PROGRAM C_Machine_CTRL
VAR
	
	bFirstRun					:BOOL;
	bFirstAutoCycle				:BOOL;
	bSmacDone					:BOOL;
	bKistlerDone				:BOOL;
	rSmacDone					:R_TRIG;
	rKistlerDone				:R_TRIG;
	bStatisticsFlag				:ARRAY[0..1] OF BOOL;
	
	eMachineState				:E_MachineState:=E_MachineState.SYSTEM_POWER_UP;

	//Timers && Triggers
	tonSys_Init					:Tc2_Standard.TON:=(PT:=T#1S);
	tonSys_InitTimeout			:Tc2_Standard.TON:=(PT:=T#3M);					
	tonWAIT_SMAC_KISLR			:Tc2_Standard.TON;
	tonFirstAutoCycle			:Tc2_Standard.TON:=(PT:=T#500MS);
	
	//Process Cycle
	eCycleState					:E_ProcessCycle;
	stTotalReport				:ST_ProcessReport;
	bStartConditions			:BOOL;	
	tonTwoHandsTouching			:Tc2_Standard.TON;         
	bScrewPresent				: BOOL;
	bReservoirPresent			: BOOL;
	tonGrippersOpennedSignal	: TON;
	tonDelayExe					:Tc2_Standard.TON:=(PT:=T#100MS);
	rtrigResetModule			:Tc2_Standard.R_TRIG;
	rtrigProcessLogShift		:Tc2_Standard.R_TRIG;
	
	
	//Index
	idx							:INT;
	
END_VAR
//----------------------------------------------------------------------------oldschoo1

// Call for Actions

   b_Machine_Status();		//State machina 
	 c_ProcessCycle();	   //Master sequencer


//----------------------------------------------------------------*


// Process Report circular buffer
rtrigProcessLogShift(CLK:=eCycleState=E_ProcessCycle.Saving_DATA);

IF rtrigProcessLogShift.Q THEN 
	FOR idx:= 250 TO 2 BY -1 DO
		GVL_PERSISTENT.stProccessReportLog[idx]:=GVL_PERSISTENT.stProccessReportLog[idx-1];
	END_FOR
	GVL_PERSISTENT.stProccessReportLog[1]:=stTotalReport;
END_IF//																										||
//--------------------------------------------------------------------------------------------------------oldschoo1

ACTION b_Machine_Status:




//Timers && Triggers
tonSys_Init(IN:=stMachineStatus.bInitialising);
tonSys_InitTimeout(IN:=stMachineStatus.bInitialising);
IF stMachineStatus.eMachineState <> E_MachineState.SYSTEM_AUTO_CYCLE THEN
	bFirstAutoCycle							:= FALSE;
END_IF

//Transition IF Cycle Stop Fault OR Imediate Fault
IF NOT stMasterCtrl.bNoMachineImmediateFault THEN		
				stMachineStatus.eMachineState := E_MachineState.IMMEDIATE_FAULT;
	
ELSIF NOT stMasterCtrl.bNoCycleStopFault AND NOT stMachineStatus.bImmediateStopped THEN
				stMachineStatus.eMachineState := E_MachineState.CYCLE_STOP_FAULT;
END_IF

IF NOT GVL_Master.stMasterCTRL.bManualModeRequest THEN
	CMD_Axis.bManualMode	:=FALSE;
	CMD_Smac.bManualMode	:=FALSE;
	CMD_Kistler.bManualMode	:=FALSE;
END_IF
(****************************************************MACHINE_CTRL*******************************************************************)
//STATE MACHINE: ------------------------------------------------------------------------------------------------------------------SM
CASE stMachineStatus.eMachineState OF

E_MachineState.SYSTEM_POWER_UP: 		// ------------------------------------------------------------------------------POWER_UP

				IF tonSystemPowerUP.Q THEN
						stMachineStatus.eMachineState := E_MachineState.IMMEDIATE_STOPPED;//
				END_IF
	
E_MachineState.IMMEDIATE_STOPPED:		// ---------------------------------------------------------------------IMMEDIATE_STOPPED

				IF stMasterCtrl.bNoMachineImmediateFault AND bResetButtonFallingEdge THEN
						stMachineStatus.eMachineState := E_MachineState.SYSTEM_INITIALISING;//
						
				ELSIF NOT stMasterCtrl.bNoCycleStopFault THEN
						stMachineStatus.eMachineState := E_MachineState.CYCLE_STOP_FAULT;//
					
				ELSIF NOT stMasterCtrl.bNoMachineImmediateFault THEN
					stMachineStatus.eMachineState := E_MachineState.IMMEDIATE_FAULT;//	
				END_IF		


E_MachineState.SYSTEM_INITIALISING:		// -------------------------------------------------------------------SYSTEM_INITIALISING		

				IF tonSys_Init.Q THEN
						CMD_Axis.bEnable	:=TRUE;
						CMD_Smac.bEnable	:=TRUE;
						CMD_Kistler.bEnable	:=TRUE;
						
						CMD_Axis.bAbort		:=FALSE;
						CMD_Smac.bAbort		:=FALSE;
						CMD_Kistler.bAbort	:=FALSE;
				END_IF

				//IF Axis_STATUS.bReady AND Kistler_STATUS.bReady  AND Smac_STATUS.bReady THEN 
				 IF Axis_STATUS.bReady AND Kistler_STATUS.bReady AND ( GVL_PERSISTENT.bSMACEnable AND Smac_STATUS.bReady OR NOT GVL_PERSISTENT.bSMACEnable) THEN //**LAA  29092025
										stMachineStatus.eMachineState:= E_MachineState.SYSTEM_READY_TO_START;//
				END_IF

				IF bStopButtonFallingEdge OR 
			 	  (stMasterCtrl.bNoMachineImmediateFault AND 
			 	  (stMasterCtrl.bCycleStopRequest OR tonSys_InitTimeout.Q) AND 
			       stMasterCtrl.bAllActionsStopped)
					THEN
										stMachineStatus.eMachineState := E_MachineState.CYCLE_STOPPED;//
						
				ELSIF stMasterCtrl.bNoMachineImmediateFault AND NOT stMasterCtrl.bNoCycleStopFault 
					THEN		
										stMachineStatus.eMachineState := E_MachineState.CYCLE_STOP_FAULT;//
			
				ELSIF NOT stMasterCtrl.bNoMachineImmediateFault 
					THEN
										stMachineStatus.eMachineState := E_MachineState.IMMEDIATE_FAULT;//
				END_IF
			
					
E_MachineState.SYSTEM_READY_TO_START:	// -------------------------------------------------------------------SYSTEM_READY_TO_START<<<

				IF 	 bStartButtonFallingEdge AND stMasterCtrl.bAllModulesReady THEN
					
										stMachineStatus.eMachineState := E_MachineState.SYSTEM_AUTO_CYCLE;//
				
				ELSIF bStopButtonFallingEdge THEN
					
										stMachineStatus.eMachineState := E_MachineState.STOPPING;//
										
				ELSIF stMasterCtrl.bNoMachineImmediateFault AND NOT stMasterCtrl.bNoCycleStopFault THEN	
	
										stMachineStatus.eMachineState := E_MachineState.CYCLE_STOP_FAULT;//
			
				ELSIF NOT stMasterCtrl.bNoMachineImmediateFault THEN
										stMachineStatus.eMachineState := E_MachineState.IMMEDIATE_FAULT;//
				ELSIF GVL_Master.stMasterCTRL.bManualModeRequest AND stMasterCtrl.bNoMachineImmediateFault AND stMasterCtrl.bNoCycleStopFault THEN
										stMachineStatus.eMachineState := E_MachineState.MANUAL_MODE;//
				END_IF

				

E_MachineState.SYSTEM_AUTO_CYCLE:		// ---------------------------------------------------------------------SYSTEM_AUTO_CYCLE	

				IF bStopButtonFallingEdge THEN					
										stMachineStatus.eMachineState := E_MachineState.STOPPING;//
						
				ELSIF stMasterCtrl.bCycleStopRequest THEN 
					
										stMachineStatus.eMachineState := E_MachineState.STOPPING;//
										
				ELSIF stMasterCtrl.bNoMachineImmediateFault AND NOT stMasterCtrl.bNoCycleStopFault THEN	
	
										stMachineStatus.eMachineState := E_MachineState.CYCLE_STOP_FAULT;//
			
				ELSIF NOT stMasterCtrl.bNoMachineImmediateFault THEN
										stMachineStatus.eMachineState := E_MachineState.IMMEDIATE_FAULT;//
				END_IF	

E_MachineState.SYSTEM_STANDBY:;//



E_MachineState.STOPPING:				// ------------------------------------------------------------------------------STOPPING

				IF stMasterCtrl.bAllActionsStopped THEN
										stMachineStatus.eMachineState := E_MachineState.CYCLE_STOPPED;//					
				END_IF
				CMD_Axis.bEnable	:=FALSE;
				CMD_Smac.bEnable	:=FALSE;
				CMD_Kistler.bEnable	:=FALSE;
				
				CMD_Axis.bAbort		:=TRUE;
				CMD_Smac.bAbort		:=TRUE;
				CMD_Kistler.bAbort	:=TRUE;

E_MachineState.CYCLE_STOPPED:			// -------------------------------------------------------------------------CYCLE_STOPPED

				IF stMasterCtrl.bNoCycleStopFault   AND 
	      		NOT stMasterCtrl.bCycleStopRequest  AND 
                               bResetButtonFallingEdge

									THEN	
										stMachineStatus.eMachineState := E_MachineState.SYSTEM_INITIALISING;		
				END_IF	

E_MachineState.IMMEDIATE_FAULT:			// -----------------------------------------------------------------------IMMEDIATE_FAULT
				
				CMD_Axis.bEnable	:=FALSE;
				CMD_Smac.bEnable	:=FALSE;
				CMD_Kistler.bEnable	:=FALSE;
						
				CMD_Axis.bAbort		:=TRUE;
				CMD_Smac.bAbort		:=TRUE;
				CMD_Kistler.bAbort	:=TRUE;
				
				IF stMasterCtrl.bNoMachineImmediateFault	THEN
										stMachineStatus.eMachineState := E_MachineState.IMMEDIATE_STOPPED;		
				END_IF

E_MachineState.CYCLE_STOP_FAULT:		// ----------------------------------------------------------------------CYCLE_STOP_FAULT

				CMD_Axis.bEnable	:=FALSE;
				CMD_Smac.bEnable	:=FALSE;
				CMD_Kistler.bEnable	:=FALSE;
						
				CMD_Axis.bAbort		:=TRUE;
				CMD_Smac.bAbort		:=TRUE;
				CMD_Kistler.bAbort	:=TRUE;
				
				IF stMasterCtrl.bNoCycleStopFault THEN
										stMachineStatus.eMachineState := E_MachineState.CYCLE_STOPPED;
				END_IF	


E_MachineState.MANUAL_MODE:;//

				IF bStopButtonFallingEdge OR NOT GVL_Master.stMasterCTRL.bManualModeRequest THEN
					
										stMachineStatus.eMachineState := E_MachineState.STOPPING;//
										
										CMD_Axis.bManualMode:=FALSE;
										CMD_Smac.bManualMode:=FALSE;
										CMD_Kistler.bManualMode:=FALSE;
										CMD_Axis.bAbort		:=TRUE;
										CMD_Smac.bAbort		:=TRUE;
										CMD_Kistler.bAbort	:=TRUE;
				ELSIF stMasterCtrl.bNoMachineImmediateFault AND NOT stMasterCtrl.bNoCycleStopFault THEN	
	
										stMachineStatus.eMachineState := E_MachineState.CYCLE_STOP_FAULT;//
										
										CMD_Axis.bManualMode:=FALSE;
										CMD_Smac.bManualMode:=FALSE;
										CMD_Kistler.bManualMode:=FALSE;
										CMD_Axis.bAbort		:=TRUE;
										CMD_Smac.bAbort		:=TRUE;
										CMD_Kistler.bAbort	:=TRUE;
			
				ELSIF NOT stMasterCtrl.bNoMachineImmediateFault THEN
							
										stMachineStatus.eMachineState := E_MachineState.IMMEDIATE_FAULT;//
				
										CMD_Axis.bManualMode:=FALSE;
										CMD_Smac.bManualMode:=FALSE;
										CMD_Kistler.bManualMode:=FALSE;
										CMD_Axis.bAbort		:=TRUE;
										CMD_Smac.bAbort		:=TRUE;
										CMD_Kistler.bAbort	:=TRUE;
										
				ELSE 					CMD_Axis.bManualMode:=TRUE;
										CMD_Smac.bManualMode:=TRUE;
										CMD_Kistler.bManualMode:=TRUE;
				END_IF
ELSE
stMachineStatus.eMachineState:=E_MachineState.SYSTEM_POWER_UP;		
END_CASE									// ------------------------------------------------------------------------------- END SM


(******************************************************MACHINE_STATUS***************************************************************)
// Status Flags -----------------------------------------------------------------------------------------------------STATUS_FLAGS
stMachineStatus.bSystemPowerUp 			:= (stMachineStatus.eMachineState = E_MachineState.SYSTEM_POWER_UP);
stMachineStatus.bImmediateStopped 		:= (stMachineStatus.eMachineState = E_MachineState.IMMEDIATE_STOPPED);
stMachineStatus.bInitialising 			:= (stMachineStatus.eMachineState = E_MachineState.SYSTEM_INITIALISING);
stMachineStatus.bReadyToStart 			:= (stMachineStatus.eMachineState = E_MachineState.SYSTEM_READY_TO_START);
stMachineStatus.bAutoCycle 				:= (stMachineStatus.eMachineState = E_MachineState.SYSTEM_AUTO_CYCLE);
stMachineStatus.bStandby 				:= (stMachineStatus.eMachineState = E_MachineState.SYSTEM_STANDBY);
stMachineStatus.bStopping 				:= (stMachineStatus.eMachineState = E_MachineState.STOPPING);
stMachineStatus.bCycleStopped 			:= (stMachineStatus.eMachineState = E_MachineState.CYCLE_STOPPED);
stMachineStatus.bImmediateFault 		:= (stMachineStatus.eMachineState = E_MachineState.IMMEDIATE_FAULT);
stMachineStatus.bCycleStopFault 		:= (stMachineStatus.eMachineState = E_MachineState.CYCLE_STOP_FAULT);
stMachineStatus.bManualMode 			:= (stMachineStatus.eMachineState = E_MachineState.MANUAL_MODE);

//Transition Flags -----------------------------------------------------------------------------------------------TRANZITION_FLAGS
stMasterCtrl.bAllActionsStopped			:= (Axis_STATUS.bReady AND Kistler_STATUS.bReady AND ( GVL_PERSISTENT.bSMACEnable AND Smac_STATUS.bReady OR NOT GVL_PERSISTENT.bSMACEnable) ) OR  //**LAA 29092025
										   (NOT Axis_STATUS.bBusy AND NOT Kistler_STATUS.bBusy );
										   
stMasterCtrl.bAllModulesReady			:= (Axis_STATUS.bReady AND Kistler_STATUS.bReady AND ( GVL_PERSISTENT.bSMACEnable AND Smac_STATUS.bReady OR NOT GVL_PERSISTENT.bSMACEnable)); //**LAA 29092025

(*stMasterCtrl.bAllActionsStopped			:= (Axis_STATUS.bReady AND Kistler_STATUS.bReady AND Smac_STATUS.bReady ) OR
										   (NOT Axis_STATUS.bBusy AND NOT Kistler_STATUS.bBusy );
										   
stMasterCtrl.bAllModulesReady			:= (Axis_STATUS.bReady AND Kistler_STATUS.bReady AND Smac_STATUS.bReady ); 

*)
END_ACTION

ACTION c_ProcessCycle:
//Timers
tonDelayExe(IN:=(eCycleState=E_ProcessCycle.AXIS_HOME AND Axis_STATUS.bReady) OR
				(eCycleState=E_ProcessCycle.AXIS_CMD_1 AND Axis_STATUS.bReady) OR
				(eCycleState=E_ProcessCycle.AXIS_CMD_2 AND Axis_STATUS.bReady) OR
				(eCycleState=E_ProcessCycle.AXIS_CMD_3 AND Axis_STATUS.bReady) OR
				(eCycleState=E_ProcessCycle.SMAC_CMD_1 AND Smac_STATUS.bReady) OR
				((eCycleState=E_ProcessCycle.CMD_SMAC_KISLR OR eCycleState=E_ProcessCycle.CMD_KISLR )AND (CMD_Kistler.bExecute OR NOT bReservoir_Present)AND (GVL_PERSISTENT.bSMACEnable AND CMD_Smac.bExecute OR NOT bScrewPresent ))
);  //AND Smac_STATUS.bReady));				//to finish
				
tonGrippersOpennedSignal( IN :=  NOT stSmac.bGripperA_ClosedSensor AND NOT stSmac.bGripperA_ClosedSensor, PT := T#1S);
tonWAIT_SMAC_KISLR(IN := eCycleState = E_ProcessCycle.WAIT_SMAC_KISLR,PT := T#500MS);
tonFirstAutoCycle( IN := eCycleState = E_ProcessCycle.IDLE AND stMachineStatus.bAutoCycle);
(******************************************************START CONDITIONS******************************************************)				
// Start Conditions: 
// - Optional add HMI PopUp if Pack fixture is in but NOT all 3 parts present -	
		
tonTwoHandsTouching(IN:=stSafety.bTwoHands_Signal, PT:=T#500MS);       // **LAA 03/12/2025 > it was too slow PT:=T#2S);

bStartConditions 		 := (tonTwoHandsTouching.Q AND 
							stMachineStatus.bAutoCycle AND
							GVL_MASTER.bPuck_Present);
							//AND bGearBox_Present 
					
							
//Reset Module --------------------------------------------------------------------------------------------------------------*
IF bResetButtonRisingEdge OR 
stMachineStatus.bCycleStopFault OR stMachineStatus.bImmediateFault OR stMachineStatus.bImmediateStopped
THEN eCycleState:=E_ProcessCycle.RESET_ALL_CMD;END_IF
//KISTLER / SMAC DONE---------------------------------------------------------------------------------------------------------*
rSmacDone( CLK := Smac_STATUS.bDone );					
rKistlerDone( CLK := Kistler_STATUS.bDone );					

IF rKistlerDone.Q THEN 
	bKistlerDone		:= TRUE;
END_IF
IF rSmacDone.Q THEN
	bSmacDone			:= TRUE;
END_IF

(************************************************************CTRL*************************************************************)
//STATE MACHINE: -----------------------------------------------------------------------------------------------------------SM
CASE eCycleState OF
						(****************************************************************IDLE********************************)
E_ProcessCycle.IDLE:	//-----------------------------------------------------------------------------------------------IDLE
									IF bStartConditions AND GVL_PERSISTENT.bSMACEnable THEN   //**LAA 29092025
										eCycleState:=E_ProcessCycle.AXIS_CMD_1;
										stTotalReport.bKis_Pass								:= FALSE;
										stTotalReport.bKis_Fail								:= FALSE;
										stTotalReport.bSmac_Pass							:= FALSE;
										stTotalReport.bSmac_Fail							:= FALSE;
										GVL_IO.qCycleIndicator_RedLED						:= FALSE;
										GVL_IO.qCycleIndicator_GreenLED						:= FALSE;
										S_Master_SMAC.bCloseGripper							:= FALSE;
										ELSIF bStartConditions AND NOT GVL_PERSISTENT.bSMACEnable THEN // *LAA  29092025
											eCycleState:=E_ProcessCycle.AXIS_CMD_2;
											stTotalReport.bKis_Pass								:= FALSE;
											stTotalReport.bKis_Fail								:= FALSE;
											stTotalReport.bSmac_Pass							:= FALSE;
											stTotalReport.bSmac_Fail							:= FALSE;
											GVL_IO.qCycleIndicator_RedLED						:= FALSE;
											GVL_IO.qCycleIndicator_GreenLED						:= FALSE;
											S_Master_SMAC.bCloseGripper							:= FALSE;
									END_IF
									 IF NOT bFirstAutoCycle AND GVL_MASTER.bPuck_Present AND
										NOT tonFirstAutoCycle.Q AND stMachineStatus.bAutoCycle THEN
										eCycleState:=E_ProcessCycle.AXIS_CMD_3;
										stTotalReport.bKis_Pass								:= FALSE;
										stTotalReport.bKis_Fail								:= FALSE;
										stTotalReport.bSmac_Pass							:= FALSE;
										stTotalReport.bSmac_Fail							:= FALSE;
										GVL_IO.qCycleIndicator_RedLED						:= FALSE;
										GVL_IO.qCycleIndicator_GreenLED						:= FALSE;
										S_Master_SMAC.bCloseGripper							:= FALSE;
									END_IF
									//Just Idleing like chilling here
									CMD_Smac.bFixtureGripper		:= FALSE;
									CMD_Smac.bGuideGripper			:= FALSE;
									IF stMachineStatus.bAutoCycle AND NOT GVL_MASTER.bPuck_Present THEN
										GVL_HMI.sMessageToOperator	:='Insert Nest';
									ELSIF stMachineStatus.bAutoCycle AND GVL_MASTER.bPuck_Present THEN
										GVL_HMI.sMessageToOperator	:='Put two hands to start Cycle Process';
									ELSIF NOT stMachineStatus.bAutoCycle AND  stMachineStatus.bReadyToStart THEN
									GVL_HMI.sMessageToOperator	:='Press START to Begin';
									ELSIF NOT stMachineStatus.bAutoCycle AND  NOT stMachineStatus.bReadyToStart THEN
									GVL_HMI.sMessageToOperator	:='Press RESET';
									END_IF
									
							(************************************************************CYCLE******************************)									
E_ProcessCycle.AXIS_CMD_1:	//-------------------------------------------------------------------------------------AXIS_CMD_1

									IF Axis_STATUS.bReady THEN
											stY_Axis.bSetToPosition[1]	:=TRUE;
									END_IF

									IF tonDelayExe.Q THEN
											CMD_Axis.bExecute			:=TRUE;
											eCycleState:=E_ProcessCycle.WAIT_AXIS_CMD_1;
									END_IF
									GVL_HMI.sMessageToOperator	:='Axis Y Moving to Position 1';
									bFirstAutoCycle						:=TRUE;
									
	
E_ProcessCycle.WAIT_AXIS_CMD_1:	//----------------------------------------------------------------------------WAIT_AXIS_CMD_1
							 		IF GVL_PERSISTENT.bSMACEnable AND Axis_STATUS.bDone AND bScrew_Present THEN
											stY_Axis.bSetToPosition[1]	:=FALSE;
											CMD_Axis.bExecute			:=FALSE;
											bScrewPresent				:=TRUE;
											eCycleState:=E_ProcessCycle.SMAC_CMD_1;
									ELSIF  GVL_PERSISTENT.bSMACEnable AND Axis_STATUS.bDone AND NOT bScrew_Present OR NOT GVL_PERSISTENT.bSMACEnable THEN
											stY_Axis.bSetToPosition[1]	:=FALSE;
											CMD_Axis.bExecute			:=FALSE;
											bScrewPresent				:=FALSE;
											eCycleState:=E_ProcessCycle.AXIS_CMD_2;
									END_IF
									
									
E_ProcessCycle.SMAC_CMD_1:	//-------------------------------------------------------------------------------------SMAC_CMD_1		//to finish
									IF  Smac_STATUS.bReady THEN
										stSmac.bSet_PickScrew				:=TRUE;
										CMD_Smac.bExecute					:=TRUE;
									END_IF
									IF  Smac_Status.bBusy THEN
										eCycleState:=E_ProcessCycle.WAIT_SMAC_CMD_1;
									END_IF
									
									GVL_HMI.sMessageToOperator	:='Smac Picking Screw Part';

	
E_ProcessCycle.WAIT_SMAC_CMD_1:	//----------------------------------------------------------------------------WAIT_SMAC_CMD_1		//to finish
									//Wait for Smac device to feedback 
									IF Smac_STATUS.bFirstPartOfCycleDone THEN
										eCycleState:=E_ProcessCycle.AXIS_CMD_2;	
										CMD_Smac.bExecute				:=FALSE;
									END_IF

E_ProcessCycle.AXIS_CMD_2:	//-------------------------------------------------------------------------------------AXIS_CMD_2
							 		
											stY_Axis.bSetToPosition[2]	:=TRUE;
									

									IF tonDelayExe.Q AND Axis_STATUS.bReady THEN
											CMD_Axis.bExecute			:=TRUE;
											eCycleState:=E_ProcessCycle.WAIT_AXIS_CMD_2;
									END_IF	
									
									GVL_HMI.sMessageToOperator	:='Axis Y Moving to Position 2';

E_ProcessCycle.WAIT_AXIS_CMD_2:	//----------------------------------------------------------------------------WAIT_AXIS_CMD_2
						 		IF Axis_STATUS.bDone  AND GVL_PERSISTENT.bSMACEnable THEN
											stY_Axis.bSetToPosition[2]	:=FALSE;
											CMD_Axis.bExecute			:=FALSE;
											eCycleState:=E_ProcessCycle.GRIPPERS_CMD_1;
											ELSIF Axis_STATUS.bDone AND NOT GVL_PERSISTENT.bSMACEnable THEN 
												stY_Axis.bSetToPosition[2]	:=FALSE;
												CMD_Axis.bExecute			:=FALSE;
												eCycleState:=E_ProcessCycle.CMD_KISLR;;
									END_IF	
E_ProcessCycle.GRIPPERS_CMD_1: //------------------------------------------------------------------------------GRIPPERS_CMD_1
								
									CMD_Smac.bFixtureGripper		:= TRUE;
									CMD_Smac.bGuideGripper			:= TRUE;
								
								eCycleState:=E_ProcessCycle.WAIT_GRIPPERS_CMD_1;
								
								

E_ProcessCycle.WAIT_GRIPPERS_CMD_1: //--------------------------------------------------------------------WAIT_GRIPPERS_CMD_1
								IF stSmac.bGripperA_ClosedSensor AND stSmac.bGripperA_ClosedSensor AND 
									(bScrewPresent OR bPuck_Present) THEN
									eCycleState:=E_ProcessCycle.CMD_SMAC_KISLR;
								ELSIF stSmac.bGripperA_ClosedSensor AND stSmac.bGripperA_ClosedSensor AND // *LAA ????????
									(bScrewPresent OR bPuck_Present) THEN
									eCycleState:=E_ProcessCycle.STORE_PROC_DATA;
								END_IF

E_ProcessCycle.CMD_SMAC_KISLR:	//-------------------------------------------------------------------------CMD_SMAC_AND_KISLR		//to finish
							 		IF Kistler_STATUS.bReady THEN // AND Smac_STATUS.bReady
											IF bReservoir_Present THEN
												CMD_Kistler.bExecute		:=TRUE;
												bReservoirPresent			:=TRUE;
											END_IF
											IF bScrewPresent THEN
											stSmac.bSet_ScrewItIn		:=TRUE;
											CMD_Smac.bExecute			:=TRUE;
											END_IF
									END_IF

									IF tonDelayExe.Q THEN
										
											eCycleState:=E_ProcessCycle.WAIT_SMAC_KISLR;
									END_IF				
									GVL_HMI.sMessageToOperator	:='Kistler and Screw Process';

E_ProcessCycle.WAIT_SMAC_KISLR:	//----------------------------------------------------------------------------WAIT_SMAC_KISLR		//to finish
						 			IF (bKistlerDone OR NOT bReservoir_Present) AND (bSmacDone OR NOT bScrewPresent) THEN
											CMD_Kistler.bExecute		:=FALSE;
											stSmac.bSet_ScrewItIn		:=FALSE;
											CMD_Smac.bExecute			:=FALSE;
											//open guide gripper
											eCycleState:=E_ProcessCycle.STORE_PROC_DATA;
									END_IF	
//**************************************LAA******************************************************************//			

E_ProcessCycle.CMD_KISLR:	//-------------------------------------------------------------------------CMD_SMAC_AND_KISLR		//to finish
							 		IF Kistler_STATUS.bReady THEN // AND Smac_STATUS.bReady
											IF bReservoir_Present THEN
												CMD_Kistler.bExecute		:=TRUE;
												bReservoirPresent			:=TRUE;
											END_IF
									END_IF

									IF tonDelayExe.Q THEN
										
											eCycleState:=E_ProcessCycle.WAIT_KISLR;
									END_IF				
									GVL_HMI.sMessageToOperator	:='Kistler processing';

E_ProcessCycle.WAIT_KISLR:	//----------------------------------------------------------------------------WAIT_SMAC_KISLR		//to finish
						 			IF (bKistlerDone OR NOT bReservoir_Present) THEN
											CMD_Kistler.bExecute		:=FALSE;
											eCycleState:=E_ProcessCycle.STORE_PROC_DATA;
									END_IF	
//**************************************LAA******************************************************************//			
E_ProcessCycle.STORE_PROC_DATA:	//----------------------------------------------------------------------------STORE_PROC_DATA		//to finish
		
	bKistlerDone 			:= FALSE;
	bSmacDone 				:= FALSE;
	
	IF bReservoirPresent THEN
		stTotalReport.bKis_Pass								:=K_Master_Kistler.stKistlerReport.bKis_Pass;
		stTotalReport.bKis_Fail								:=K_Master_Kistler.stKistlerReport.bKis_Fail;
		stTotalReport.rKis_HighestRecordedForce				:=K_Master_Kistler.stKistlerReport.rKis_HighestRecordedForce;
		stTotalReport.rKis_LowestRecordedForce				:=K_Master_Kistler.stKistlerReport.rKis_LowestRecordedForce;
		stTotalReport.rKis_DistanceRecord					:=K_Master_Kistler.stKistlerReport.rKis_DistanceRecord;
		stTotalReport.rKis_Settings_ForceUpperTreshold		:=K_Master_Kistler.stKistlerReport.rKis_Settings_ForceUpperTreshold;
		stTotalReport.rKis_Settings_ForceLowerTreshold		:=K_Master_Kistler.stKistlerReport.rKis_Settings_ForceLowerTreshold;
		stTotalReport.rKis_Settings_StartMeasurePoint		:=K_Master_Kistler.stKistlerReport.rKis_Settings_StartMeasurePoint;
		stTotalReport.rKis_Settings_ReservoirBottomPoint	:=K_Master_Kistler.stKistlerReport.rKis_Settings_ReservoirBottomPoint;
		IF stTotalReport.bKis_Pass THEN
			stTotalReport.sKis_Result							:='PASS';
		ELSIF stTotalReport.bKis_FaiL THEN
			stTotalReport.sKis_Result							:='FAIL';
		ELSE stTotalReport.sKis_Result							:='';
		END_IF
	ELSE
		stTotalReport.bKis_Pass								:=FALSE;
		stTotalReport.bKis_Fail								:=FALSE;
		stTotalReport.rKis_HighestRecordedForce				:=0;
		stTotalReport.rKis_LowestRecordedForce				:=0;
		stTotalReport.rKis_Settings_ForceUpperTreshold		:=0;
		stTotalReport.rKis_Settings_ForceLowerTreshold		:=0;
		stTotalReport.rKis_Settings_StartMeasurePoint		:=0;
		stTotalReport.rKis_Settings_ReservoirBottomPoint	:=0;
		stTotalReport.sKis_Result							:='';
	END_IF
	IF GVL_PERSISTENT.bSMACEnable AND bScrewPresent THEN
		stTotalReport.rSmac_Settings_LinearAcc				:=S_Master_SMAC.stSmacReport.rSmac_Settings_LinearAcc;
		stTotalReport.rSmac_Settings_LinearVel				:=S_Master_SMAC.stSmacReport.rSmac_Settings_LinearVel;
		stTotalReport.rSmac_Settings_RotativeAcc			:=S_Master_SMAC.stSmacReport.rSmac_Settings_RotativeAcc;
		stTotalReport.rSmac_Settings_RotativeVel			:=S_Master_SMAC.stSmacReport.rSmac_Settings_RotativeVel;
		stTotalReport.rSmac_Settings_LinearTorque			:=S_Master_SMAC.stSmacReport.rSmac_Settings_LinearTorque;
		stTotalReport.rSmac_MaxDistanceReached				:=S_Master_SMAC.stSmacReport.rSmac_MaxDistanceReached;
		stTotalReport.bSmac_Pass							:=S_Master_SMAC.stSmacReport.bSmac_Pass;
		stTotalReport.bSmac_Fail							:=S_Master_SMAC.stSmacReport.bSmac_Fail;
		IF stTotalReport.bSmac_Pass THEN
			stTotalReport.sSmac_Result							:='PASS';
		ELSIF stTotalReport.bSmac_Fail THEN
			stTotalReport.sSmac_Result							:='FAIL';
		ELSE stTotalReport.sSmac_Result							:='';
		END_IF
	ELSE
		stTotalReport.rSmac_Settings_LinearAcc				:=0;
		stTotalReport.rSmac_Settings_LinearVel				:=0;
		stTotalReport.rSmac_Settings_RotativeAcc			:=0;
		stTotalReport.rSmac_Settings_RotativeVel			:=0;
		stTotalReport.rSmac_Settings_LinearTorque			:=0;
		stTotalReport.rSmac_MaxDistanceReached				:=0;
		stTotalReport.bSmac_Pass							:=FALSE;
		stTotalReport.bSmac_Fail							:=FALSE;
		stTotalReport.sSmac_Result							:='';
	END_IF
	
	stTotalReport.sDate										:= GVL_MASTER.sSystemDate;
	stTotalReport.sTime										:= GVL_MASTER.sSystemTime;
	
	//STATISTICS
	IF bReservoirPresent AND stTotalReport.bKis_Pass AND NOT bStatisticsFlag[0] THEN
		GVL_PERSISTENT.nKistlerGoodParts					:= GVL_PERSISTENT.nKistlerGoodParts + 1;
		GVL_PERSISTENT.nKistlerTotalGoodParts				:= GVL_PERSISTENT.nKistlerTotalGoodParts + 1;
		bStatisticsFlag[0]									:= TRUE;
	END_IF
	IF bReservoirPresent AND stTotalReport.bKis_Fail AND NOT bStatisticsFlag[0] THEN
		GVL_PERSISTENT.nKistlerBadParts						:= GVL_PERSISTENT.nKistlerBadParts + 1;
		GVL_PERSISTENT.nKistlerTotalBadParts				:= GVL_PERSISTENT.nKistlerTotalBadParts + 1;
		bStatisticsFlag[0]									:= TRUE;
	END_IF
	
	IF bScrewPresent AND stTotalReport.bSmac_Pass AND NOT bStatisticsFlag[1] THEN
		GVL_PERSISTENT.nSmacGoodParts						:= GVL_PERSISTENT.nSmacGoodParts + 1;
		GVL_PERSISTENT.nSmacTotalGoodParts					:= GVL_PERSISTENT.nSmacTotalGoodParts + 1;
		bStatisticsFlag[1]									:= TRUE;
	END_IF
		IF bScrewPresent AND stTotalReport.bSmac_Fail AND NOT bStatisticsFlag[1] THEN
		GVL_PERSISTENT.nSmacBadParts						:= GVL_PERSISTENT.nSmacBadParts + 1;
		GVL_PERSISTENT.nSmacTotalBadParts					:= GVL_PERSISTENT.nSmacTotalBadParts + 1;
		bStatisticsFlag[1]									:= TRUE;
	END_IF
	
			
			
									eCycleState:=E_ProcessCycle.Saving_DATA;	
E_ProcessCycle.Saving_DATA: //------------------------------------------------------------------------------------Saving_DATA
									eCycleState:=E_ProcessCycle.GRIPPERS_CMD_2;
									bStatisticsFlag[0]									:= FALSE;
									bStatisticsFlag[1]									:= FALSE;
									IF (bReservoirPresent AND stTotalReport.bKis_Pass) OR 
										(bScrewPresent AND stTotalReport.bSmac_Pass)THEN
										GVL_IO.qCycleIndicator_GreenLED						:= TRUE;
									ELSIF (bReservoirPresent AND stTotalReport.bKis_Fail) OR 
										(bScrewPresent AND stTotalReport.bSmac_Fail) THEN
										GVL_IO.qCycleIndicator_RedLED						:= TRUE;		
									END_IF
E_ProcessCycle.GRIPPERS_CMD_2: //------------------------------------------------------------------------------GRIPPERS_CMD_1
								
								CMD_Smac.bFixtureGripper		:= FALSE;
								CMD_Smac.bGuideGripper			:= FALSE;
								
								eCycleState:=E_ProcessCycle.WAIT_GRIPPERS_CMD_2;
								
								
								

E_ProcessCycle.WAIT_GRIPPERS_CMD_2: //--------------------------------------------------------------------WAIT_GRIPPERS_CMD_1
								IF tonGrippersOpennedSignal.Q THEN
								eCycleState:=E_ProcessCycle.AXIS_CMD_3;
								END_IF
			
E_ProcessCycle.AXIS_CMD_3:	//-------------------------------------------------------------------------------------AXIS_CMD_3
						 		IF Axis_STATUS.bReady THEN
											stY_Axis.bSetToPosition[3]	:=TRUE;
									END_IF

									IF tonDelayExe.Q THEN
											CMD_Axis.bExecute			:=TRUE;
											eCycleState:=E_ProcessCycle.WAIT_AXIS_CMD_3;
									END_IF		
								GVL_HMI.sMessageToOperator	:='Take Nest please';

E_ProcessCycle.WAIT_AXIS_CMD_3:	//----------------------------------------------------------------------------WAIT_AXIS_CMD_3
							 		IF Axis_STATUS.bDone THEN
											stY_Axis.bSetToPosition[3]	:=FALSE;
											CMD_Axis.bExecute			:=FALSE;
											eCycleState:=E_ProcessCycle.AXIS_HOME;
									END_IF


E_ProcessCycle.AXIS_HOME:	//-------------------------------------------------------------------------------------AXIS_HOME
							 		IF Axis_STATUS.bReady THEN
											stY_Axis.bSetToHome			:=TRUE;
											Y_Master_Y_Axis.bRetract 	:=TRUE;
									END_IF

									IF tonDelayExe.Q THEN
											CMD_Axis.bExecute			:=TRUE;
											eCycleState:=E_ProcessCycle.WAIT_AXIS_HOME;
									END_IF
									GVL_HMI.sMessageToOperator	:='Axis Y Homing';

E_ProcessCycle.WAIT_AXIS_HOME:	//----------------------------------------------------------------------------WAIT_AXIS_HOME
							 		IF Axis_STATUS.bDone THEN
											stY_Axis.bSetToHome			:=FALSE;
											CMD_Axis.bExecute			:=FALSE;
											Y_Master_Y_Axis.bRetract 	:=FALSE;
											eCycleState:=E_ProcessCycle.IDLE;
									END_IF
									bFirstAutoCycle						:=TRUE;

									
								(*********************************************************RESET*****************************)
E_ProcessCycle.RESET_ALL_CMD:	//------------------------------------------------------------------------------RESET_ALL_CMD

											CMD_Axis.bExecute									:=FALSE;
											CMD_Smac.bExecute									:=FALSE;
											CMD_Kistler.bExecute								:=FALSE;
											
											stSmac.bSet_PickScrew								:=FALSE;											
											stSmac.bSet_ScrewItIn								:=FALSE;
											CMD_Smac.bFixtureGripper							:= FALSE;
											CMD_Smac.bGuideGripper								:= FALSE;


											stY_Axis.bSetToHome									:=FALSE;
											Y_Master_Y_Axis.bRetract 							:=FALSE;
											stY_Axis.bSetToPosition[1]							:=FALSE;
											stY_Axis.bSetToPosition[2]							:=FALSE;
											stY_Axis.bSetToPosition[3]							:=FALSE;
											
											bKistlerDone 										:= FALSE;
											bSmacDone 											:= FALSE;
											bScrewPresent										:= FALSE;
											
											
											


											eCycleState:=E_ProcessCycle.IDLE;
											
	
ELSE
eCycleState:=E_ProcessCycle.RESET_ALL_CMD;		
END_CASE	// -------------------------------------------------------------------------------------------------------- END SM

(************************************************************STATUS************************************************************)
stMachineStatus.bProcessCycle := eCycleState <> E_ProcessCycle.IDLE AND eCycleState <> E_ProcessCycle.RESET_ALL_CMD;

//---------------------------------------------------------------------------------------------------------------------oldschoo1
END_ACTION

END_PROGRAM

(* stored: Version 1.1.0.1, ProductVersion 3.1.4024.12
   POU C_Machine_CTRL: Id {1b8b0cab-1e15-45dd-abc7-e58024eda65a}, SpecialFunc None
   Action b_Machine_Status: Id {b6145e3c-946a-45ea-af33-35f0ef7a03eb}
   Action c_ProcessCycle: Id {680539a3-5409-4299-95ed-f307f3651986} *)
